PROGRAM MAIN
VAR
	
END_VAR

// Open PLC HMI view here C:\TwinCAT\3.1\Components\Plc\Tc3PlcHmi
// Open PLC HMI web view with this link   http://127.0.0.1/Tc3PlcHmiWeb/Port_851/Visu/webvisu.htm


OP_BTN();

END_PROGRAM

(* stored: Version 1.1.0.1, ProductVersion 3.1.4024.12
   POU MAIN: Id {d3c7fc20-9915-42b0-84f1-c5b81a710447}, SpecialFunc None *)
